// TIA Portal V19 export
DATA_BLOCK "PTrk"   // DB26
// stored: Access Published, MemoryReserve 100
   VAR RETAIN
      Last_P_ID : DInt;   // Ultimo ID asseggnato a una parte (Part/Semi-guscio)
   END_VAR
   VAR
      Empty : "PTrk_Item";
   END_VAR
   VAR RETAIN
      A0202 : Struct
         Empty : Bool;
         Ready : Bool;
         Part_Qty : Int;
         Part_Len : Real;
         Beam_Len_Candidate : Real;
         P : Array[1.."PTRK_A0202_ITEMS"] of "PTrk_Item";   // Tracciamento SG su rulliera do accelerazione dopo la stazone di taglio profili = Semi-gusci
      END_STRUCT;
      A02_EXIT_TOCHECK : Array[1.."PTRK_A0202_EXIT_TOCHECK_ITEMS"] of "PTrk_Item";   // Tracciamento SG su scivolo di scarico da rulliera di accelerazione( Da controllare / Conformi per cico solo semi-gusci)
      A0301 : Struct
         Empty : Bool;
         Ready : Bool;
         Part_Qty : Int;
         Part_Len : Real;
         Beam_Len_Candidate : Real;
         P : Array[1.."PTRK_A0301_ITEMS"] of "PTrk_Item";   // Tracciamento SG su stazione di assemblaggio (capovolgimento dei due semi-gusci uno sopra all'altro)
      END_STRUCT;
   END_VAR
BEGIN
   // A0202.P[1] : PTRK_A0202_CUTTED
   // A0202.P[2] : PTRK_A0202_ENTRY
   // A0202.P[3] : PTRK_A0202_P6
   // A0202.P[4] : PTRK_A0202_P5
   // A0202.P[5] : PTRK_A0202_P4
   // A0202.P[6] : PTRK_A0202_P3
   // A0202.P[7] : PTRK_A0202_P2
   // A0202.P[8] : PTRK_A0202_P1
   // A0202.P[9] : PTRK_A02_S2_P0
   // A0202.P[10] : PTRK_A0202_DEVIATOR_To_A0301
   // A0202.P[11] : PTRK_A0202_DEVITATOR_To_EXIT
   // A0202.P[12] : Free
   // A0202.P[13] : Free
   // A0202.P[14] : Free
   // A0202.P[15] : Free
   // A02_EXIT_TOCHECK[1] : Ultimo SG deviato
END_DATA_BLOCK
